PROGRAM MAIN
VAR
	nRawAnalogInput : INT;
	fMotorSpeedPercent: REAL;
END_VAR

IF nRawAnalogInput < 0 THEN
	nRawAnalogInput :=0;
	
ELSIF nRawAnalogInput > 32767 THEN
	nRawAnalogInput := 32767;
END_IF

fMotorSpeedPercent := (INT_TO_REAL(nRawAnalogInput)/32767.0)*100.0;

END_PROGRAM

(* stored: Version 1.1.0.1
   POU MAIN: Id {336c7725-c845-452d-b520-242298a68d82}, SpecialFunc None *)
